// TIA Portal V19 export
FUNCTION "FC903_SafetyOutputs" : Void   // FC903, F_LAD
{ S7_Optimized_Access := 'TRUE' }
// stored: AutoNumber false
BEGIN

REGION Network 1: Open Z Axis brake
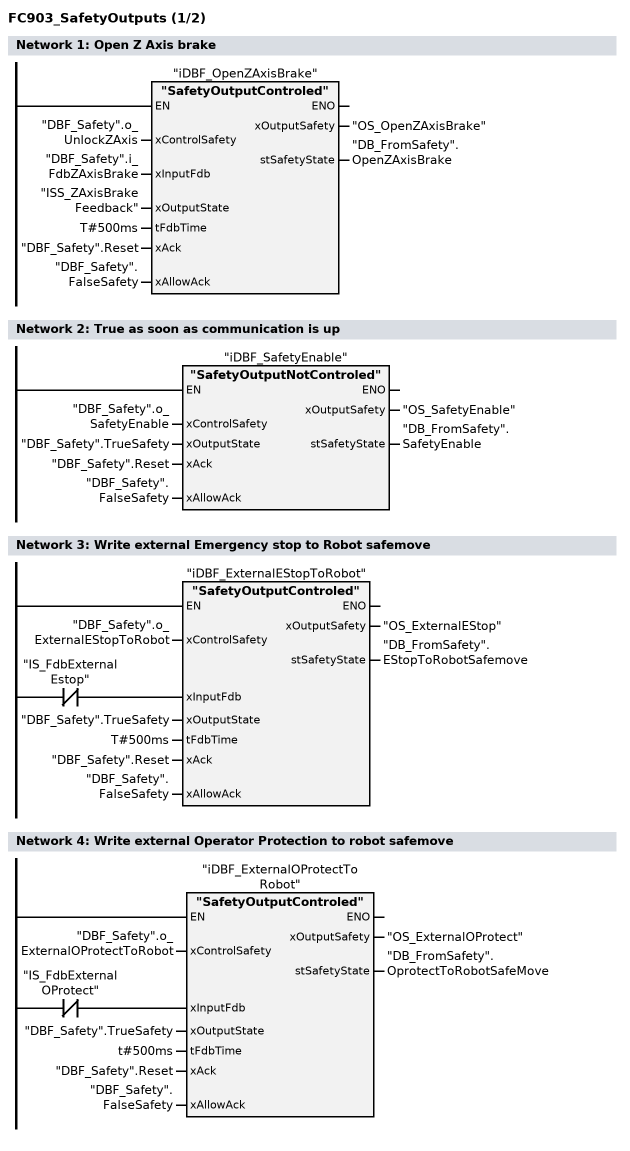
   RUNG wire#powerrail
      "iDBF_OpenZAxisBrake"(xControlSafety := "DBF_Safety".o_UnlockZAxis, xInputFdb := "DBF_Safety".i_FdbZAxisBrake, xOutputState := "ISS_ZAxisBrakeFeedback", tFdbTime := T#500ms, xAck := "DBF_Safety".Reset, xAllowAck := "DBF_Safety".FalseSafety, xOutputSafety => "OS_OpenZAxisBrake", stSafetyState => "DB_FromSafety".OpenZAxisBrake)
   END_RUNG
   // the same network as SCL:
   "iDBF_OpenZAxisBrake"(xControlSafety := "DBF_Safety".o_UnlockZAxis,   // "SafetyOutputControled"
                         xInputFdb := "DBF_Safety".i_FdbZAxisBrake,
                         xOutputState := "ISS_ZAxisBrakeFeedback",
                         tFdbTime := T#500ms,
                         xAck := "DBF_Safety".Reset,
                         xAllowAck := "DBF_Safety".FalseSafety,
                         xOutputSafety => "OS_OpenZAxisBrake",
                         stSafetyState => "DB_FromSafety".OpenZAxisBrake);
END_REGION

REGION Network 2: True as soon as communication is up
   RUNG wire#powerrail
      "iDBF_SafetyEnable"(xControlSafety := "DBF_Safety".o_SafetyEnable, xOutputState := "DBF_Safety".TrueSafety, xAck := "DBF_Safety".Reset, xAllowAck := "DBF_Safety".FalseSafety, xOutputSafety => "OS_SafetyEnable", stSafetyState => "DB_FromSafety".SafetyEnable)
   END_RUNG
   // the same network as SCL:
   "iDBF_SafetyEnable"(xControlSafety := "DBF_Safety".o_SafetyEnable,   // "SafetyOutputNotControled"
                       xOutputState := "DBF_Safety".TrueSafety,
                       xAck := "DBF_Safety".Reset,
                       xAllowAck := "DBF_Safety".FalseSafety,
                       xOutputSafety => "OS_SafetyEnable",
                       stSafetyState => "DB_FromSafety".SafetyEnable);
END_REGION

REGION Network 3: Write external Emergency stop to Robot safemove
   RUNG wire#powerrail
      "iDBF_ExternalEStopToRobot"(xInputFdb := wire#w1, xControlSafety := "DBF_Safety".o_ExternalEStopToRobot, xOutputState := "DBF_Safety".TrueSafety, tFdbTime := T#500ms, xAck := "DBF_Safety".Reset, xAllowAck := "DBF_Safety".FalseSafety, xOutputSafety => "OS_ExternalEStop", stSafetyState => "DB_FromSafety".EStopToRobotSafemove)
   END_RUNG
   RUNG wire#powerrail
      I_Contact( "IS_FdbExternalEstop" )
   END_RUNG wire#w1
   // the same network as SCL:
   "iDBF_ExternalEStopToRobot"(xControlSafety := "DBF_Safety".o_ExternalEStopToRobot,   // "SafetyOutputControled"
                           xInputFdb := NOT "IS_FdbExternalEstop",
                           xOutputState := "DBF_Safety".TrueSafety,
                           tFdbTime := T#500ms,
                           xAck := "DBF_Safety".Reset,
                           xAllowAck := "DBF_Safety".FalseSafety,
                           xOutputSafety => "OS_ExternalEStop",
                           stSafetyState => "DB_FromSafety".EStopToRobotSafemove);
END_REGION

REGION Network 4: Write external Operator Protection to robot safemove
   RUNG wire#powerrail
      "iDBF_ExternalOProtectToRobot"(xInputFdb := wire#w1, xControlSafety := "DBF_Safety".o_ExternalOProtectToRobot, xOutputState := "DBF_Safety".TrueSafety, tFdbTime := t#500ms, xAck := "DBF_Safety".Reset, xAllowAck := "DBF_Safety".FalseSafety, xOutputSafety => "OS_ExternalOProtect", stSafetyState => "DB_FromSafety".OprotectToRobotSafeMove)
   END_RUNG
   RUNG wire#powerrail
      I_Contact( "IS_FdbExternalOProtect" )
   END_RUNG wire#w1
   // the same network as SCL:
   "iDBF_ExternalOProtectToRobot"(xControlSafety := "DBF_Safety".o_ExternalOProtectToRobot,   // "SafetyOutputControled"
                           xInputFdb := NOT "IS_FdbExternalOProtect",
                           xOutputState := "DBF_Safety".TrueSafety,
                           tFdbTime := t#500ms,
                           xAck := "DBF_Safety".Reset,
                           xAllowAck := "DBF_Safety".FalseSafety,
                           xOutputSafety => "OS_ExternalOProtect",
                           stSafetyState => "DB_FromSafety".OprotectToRobotSafeMove);
END_REGION

REGION Network 5: Power Off 24V safety for FerRobotic Head
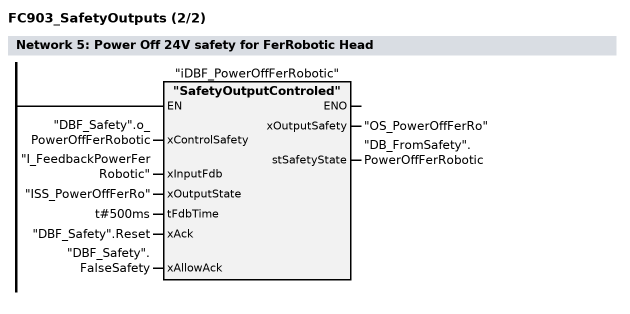
   RUNG wire#powerrail
      "iDBF_PowerOffFerRobotic"(xControlSafety := "DBF_Safety".o_PowerOffFerRobotic, xInputFdb := "I_FeedbackPowerFerRobotic", xOutputState := "ISS_PowerOffFerRo", tFdbTime := t#500ms, xAck := "DBF_Safety".Reset, xAllowAck := "DBF_Safety".FalseSafety, xOutputSafety => "OS_PowerOffFerRo", stSafetyState => "DB_FromSafety".PowerOffFerRobotic)
   END_RUNG
   // the same network as SCL:
   "iDBF_PowerOffFerRobotic"(xControlSafety := "DBF_Safety".o_PowerOffFerRobotic,   // "SafetyOutputControled"
                           xInputFdb := "I_FeedbackPowerFerRobotic",
                           xOutputState := "ISS_PowerOffFerRo",
                           tFdbTime := t#500ms,
                           xAck := "DBF_Safety".Reset,
                           xAllowAck := "DBF_Safety".FalseSafety,
                           xOutputSafety => "OS_PowerOffFerRo",
                           stSafetyState => "DB_FromSafety".PowerOffFerRobotic);
END_REGION
END_FUNCTION
